PROGRAM PRG_TEST
VAR
	//fbCaseDuplicatCheckTests			: FB_CASE_DuplicatCheckTests;
	//fbCaseDuplicateUpdateToDBTests	: FB_CASE_DuplicateUpdateToDBTests;
	//fbCaseFinaliseDataTests				: FB_CASE_FinaliseDataTests;
	//fbCaseInitialiseData_Test 			: FB_CASE_InitialiseDataTests;
	fbCaseValidateContentTests		: FB_CASE_ValidateContentTests;
	
END_VAR

//===================================================
//UNIT TEST EXECUTION

TcUnit.RUN();

//===================================================
//MANUAL TEST EXECUTION

PRG_CASE_DuplicatCheckManual();
PRG_CASE_DuplicateUpdateToDBManual();
PRG_CASE_FinaliseDataManual();
PRG_CASE_InitialiseDataManual();
PRG_CASE_ValidateContentManual();



//===================================================
//TESTS for FB references
//PRG_Reference_POU();

END_PROGRAM

(* stored: Version 1.1.0.1
   POU PRG_TEST: Id {57de771e-4346-4079-9379-3645d39749ca}, SpecialFunc None *)
